{attribute 'qualified_only'}
VAR_GLOBAL
	button_pressed : BOOL;
	lamp_on : BOOL;
END_VAR

(* stored: Version 1.1.0.1, ProductVersion 3.1.4024.12
   GVL GVL: Id {c54b9728-225c-4ba4-ae73-b59ee8cd2aac} *)
